Staubli VAL3: dataListAdd.pgx

program dataListAdd(string x_sEvent)
begin
  // add in the queue
  if sDataList!=""
    insert(sDataList[size(sDataList)])
  endIf
  sDataList[size(sDataList)-1]=x_sEvent
end
